// TIA Portal V20 export
FUNCTION_BLOCK "FB Equipment Modules"   // FB2, LAD
TITLE = FB - Equipment Modules
{ S7_Optimized_Access := 'TRUE' }
// stored: MemoryReserve 100, SetENOAutomatically false
   VAR
      "Instance - Bas342" { S7_SetPoint := 'True'} : "FB - Bas342";
      "Instance - TableCheck - Process1" { S7_SetPoint := 'True'} : "FB - TableCheck";
      "Instance - TableCheck - Process2" { S7_SetPoint := 'True'} : "FB - TableCheck";
      "Instance - Sabload - P1 Left" { S7_SetPoint := 'True'} : "FB - Sabload";
      "Instance - Sabload - P1 Right" { S7_SetPoint := 'True'} : "FB - Sabload";
      "Instance - Sabload - P2 Left" { S7_SetPoint := 'True'} : "FB - Sabload";
      "Instance - Sabload - P2 Right" { S7_SetPoint := 'True'} : "FB - Sabload";
   END_VAR
BEGIN

REGION Network 1: Module - Bas342
   // Call of the Bas342 module.
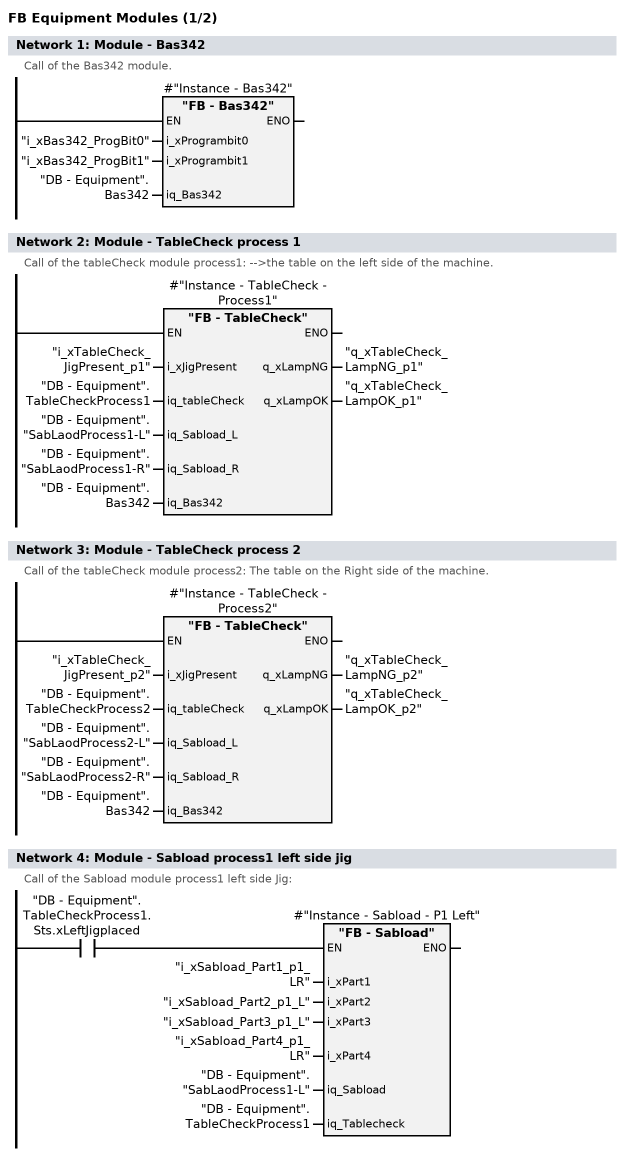
   RUNG wire#powerrail
      #"Instance - Bas342"(i_xProgrambit0 := "i_xBas342_ProgBit0", i_xProgrambit1 := "i_xBas342_ProgBit1", iq_Bas342 := "DB - Equipment".Bas342)
   END_RUNG
   // the same network as SCL:
   #"Instance - Bas342"(i_xProgrambit0 := "i_xBas342_ProgBit0",   // "FB - Bas342"
                        i_xProgrambit1 := "i_xBas342_ProgBit1",
                        iq_Bas342 := "DB - Equipment".Bas342);
END_REGION

REGION Network 2: Module - TableCheck process 1
   // Call of the tableCheck module process1: -->the table on the left side of the machine.
   RUNG wire#powerrail
      #"Instance - TableCheck - Process1"(i_xJigPresent := "i_xTableCheck_JigPresent_p1", iq_tableCheck := "DB - Equipment".TableCheckProcess1, iq_Sabload_L := "DB - Equipment"."SabLaodProcess1-L", iq_Sabload_R := "DB - Equipment"."SabLaodProcess1-R", iq_Bas342 := "DB - Equipment".Bas342, q_xLampNG => "q_xTableCheck_LampNG_p1", q_xLampOK => "q_xTableCheck_LampOK_p1")
   END_RUNG
   // the same network as SCL:
   #"Instance - TableCheck - Process1"(i_xJigPresent := "i_xTableCheck_JigPresent_p1",   // "FB - TableCheck"
                           iq_tableCheck := "DB - Equipment".TableCheckProcess1,
                           iq_Sabload_L := "DB - Equipment"."SabLaodProcess1-L",
                           iq_Sabload_R := "DB - Equipment"."SabLaodProcess1-R",
                           iq_Bas342 := "DB - Equipment".Bas342,
                           q_xLampNG => "q_xTableCheck_LampNG_p1",
                           q_xLampOK => "q_xTableCheck_LampOK_p1");
END_REGION

REGION Network 3: Module - TableCheck process 2
   // Call of the tableCheck module process2: The table on the Right side of the machine.
   RUNG wire#powerrail
      #"Instance - TableCheck - Process2"(i_xJigPresent := "i_xTableCheck_JigPresent_p2", iq_tableCheck := "DB - Equipment".TableCheckProcess2, iq_Sabload_L := "DB - Equipment"."SabLaodProcess2-L", iq_Sabload_R := "DB - Equipment"."SabLaodProcess2-R", iq_Bas342 := "DB - Equipment".Bas342, q_xLampNG => "q_xTableCheck_LampNG_p2", q_xLampOK => "q_xTableCheck_LampOK_p2")
   END_RUNG
   // the same network as SCL:
   #"Instance - TableCheck - Process2"(i_xJigPresent := "i_xTableCheck_JigPresent_p2",   // "FB - TableCheck"
                           iq_tableCheck := "DB - Equipment".TableCheckProcess2,
                           iq_Sabload_L := "DB - Equipment"."SabLaodProcess2-L",
                           iq_Sabload_R := "DB - Equipment"."SabLaodProcess2-R",
                           iq_Bas342 := "DB - Equipment".Bas342,
                           q_xLampNG => "q_xTableCheck_LampNG_p2",
                           q_xLampOK => "q_xTableCheck_LampOK_p2");
END_REGION

REGION Network 4: Module - Sabload process1 left side jig
   // Call of the Sabload module process1 left side Jig:
   RUNG wire#powerrail
      Contact( "DB - Equipment".TableCheckProcess1.Sts.xLeftJigplaced )
      #"Instance - Sabload - P1 Left"(i_xPart1 := "i_xSabload_Part1_p1_LR", i_xPart2 := "i_xSabload_Part2_p1_L", i_xPart3 := "i_xSabload_Part3_p1_L", i_xPart4 := "i_xSabload_Part4_p1_LR", iq_Sabload := "DB - Equipment"."SabLaodProcess1-L", iq_Tablecheck := "DB - Equipment".TableCheckProcess1)
   END_RUNG
   // the same network as SCL:
   IF "DB - Equipment".TableCheckProcess1.Sts.xLeftJigplaced THEN
       #"Instance - Sabload - P1 Left"(i_xPart1 := "i_xSabload_Part1_p1_LR",   // "FB - Sabload"
                               i_xPart2 := "i_xSabload_Part2_p1_L",
                               i_xPart3 := "i_xSabload_Part3_p1_L",
                               i_xPart4 := "i_xSabload_Part4_p1_LR",
                               iq_Sabload := "DB - Equipment"."SabLaodProcess1-L",
                               iq_Tablecheck := "DB - Equipment".TableCheckProcess1);
   END_IF;
END_REGION

REGION Network 5: Module - Sabload process1 Right side jig
   // Call of the Sabload module process1 Right side Jig:
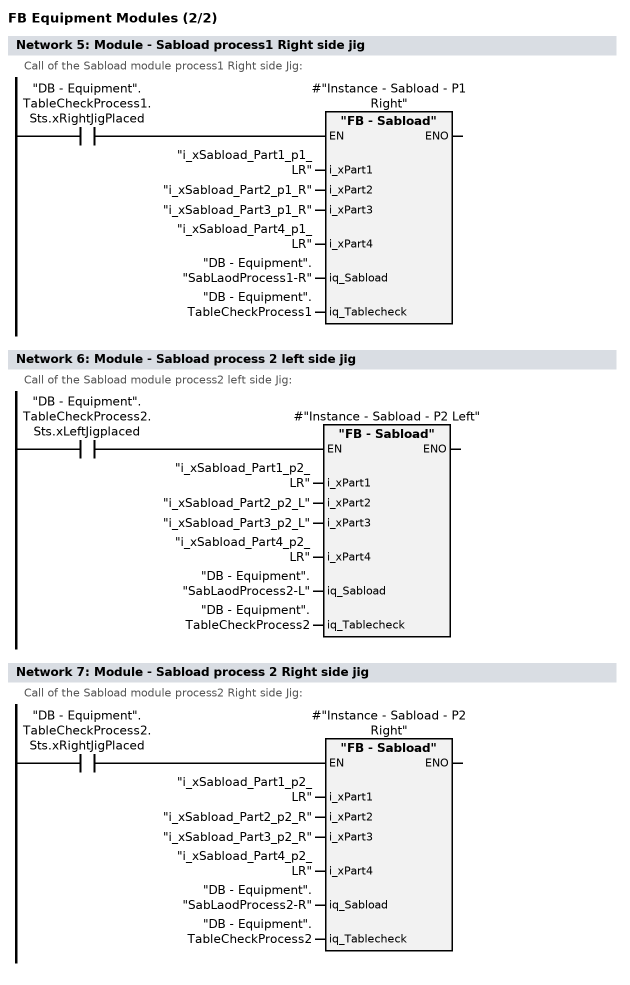
   RUNG wire#powerrail
      Contact( "DB - Equipment".TableCheckProcess1.Sts.xRightJigPlaced )
      #"Instance - Sabload - P1 Right"(i_xPart1 := "i_xSabload_Part1_p1_LR", i_xPart2 := "i_xSabload_Part2_p1_R", i_xPart3 := "i_xSabload_Part3_p1_R", i_xPart4 := "i_xSabload_Part4_p1_LR", iq_Sabload := "DB - Equipment"."SabLaodProcess1-R", iq_Tablecheck := "DB - Equipment".TableCheckProcess1)
   END_RUNG
   // the same network as SCL:
   IF "DB - Equipment".TableCheckProcess1.Sts.xRightJigPlaced THEN
       #"Instance - Sabload - P1 Right"(i_xPart1 := "i_xSabload_Part1_p1_LR",   // "FB - Sabload"
                               i_xPart2 := "i_xSabload_Part2_p1_R",
                               i_xPart3 := "i_xSabload_Part3_p1_R",
                               i_xPart4 := "i_xSabload_Part4_p1_LR",
                               iq_Sabload := "DB - Equipment"."SabLaodProcess1-R",
                               iq_Tablecheck := "DB - Equipment".TableCheckProcess1);
   END_IF;
END_REGION

REGION Network 6: Module - Sabload process 2 left side jig
   // Call of the Sabload module process2 left side Jig:
   RUNG wire#powerrail
      Contact( "DB - Equipment".TableCheckProcess2.Sts.xLeftJigplaced )
      #"Instance - Sabload - P2 Left"(i_xPart1 := "i_xSabload_Part1_p2_LR", i_xPart2 := "i_xSabload_Part2_p2_L", i_xPart3 := "i_xSabload_Part3_p2_L", i_xPart4 := "i_xSabload_Part4_p2_LR", iq_Sabload := "DB - Equipment"."SabLaodProcess2-L", iq_Tablecheck := "DB - Equipment".TableCheckProcess2)
   END_RUNG
   // the same network as SCL:
   IF "DB - Equipment".TableCheckProcess2.Sts.xLeftJigplaced THEN
       #"Instance - Sabload - P2 Left"(i_xPart1 := "i_xSabload_Part1_p2_LR",   // "FB - Sabload"
                               i_xPart2 := "i_xSabload_Part2_p2_L",
                               i_xPart3 := "i_xSabload_Part3_p2_L",
                               i_xPart4 := "i_xSabload_Part4_p2_LR",
                               iq_Sabload := "DB - Equipment"."SabLaodProcess2-L",
                               iq_Tablecheck := "DB - Equipment".TableCheckProcess2);
   END_IF;
END_REGION

REGION Network 7: Module - Sabload process 2 Right side jig
   // Call of the Sabload module process2 Right side Jig:
   RUNG wire#powerrail
      Contact( "DB - Equipment".TableCheckProcess2.Sts.xRightJigPlaced )
      #"Instance - Sabload - P2 Right"(i_xPart1 := "i_xSabload_Part1_p2_LR", i_xPart2 := "i_xSabload_Part2_p2_R", i_xPart3 := "i_xSabload_Part3_p2_R", i_xPart4 := "i_xSabload_Part4_p2_LR", iq_Sabload := "DB - Equipment"."SabLaodProcess2-R", iq_Tablecheck := "DB - Equipment".TableCheckProcess2)
   END_RUNG
   // the same network as SCL:
   IF "DB - Equipment".TableCheckProcess2.Sts.xRightJigPlaced THEN
       #"Instance - Sabload - P2 Right"(i_xPart1 := "i_xSabload_Part1_p2_LR",   // "FB - Sabload"
                               i_xPart2 := "i_xSabload_Part2_p2_R",
                               i_xPart3 := "i_xSabload_Part3_p2_R",
                               i_xPart4 := "i_xSabload_Part4_p2_LR",
                               iq_Sabload := "DB - Equipment"."SabLaodProcess2-R",
                               iq_Tablecheck := "DB - Equipment".TableCheckProcess2);
   END_IF;
END_REGION
END_FUNCTION_BLOCK
